// TIA Portal V17 export
// export: Created 2021-12-03T08:13:12.9041866Z, ExportSetting WithDefaults, DisplayName Totally Integrated Automation Portal, DisplayVersion V17, DisplayName TIA Portal Openness, DisplayVersion V17, DisplayName TIA Portal Version Control Interface, DisplayVersion V17, DisplayName STEP 7 Professional, DisplayVersion V17, DisplayName STEP 7 Safety, DisplayVersion V17, DisplayName WinCC Advanced, DisplayVersion V17
FUNCTION "FC_Safety_PerimeterCtrl" : Void   // FC300, F_FBD
VERSION : 0.1
// stored: AutoNumber false, IsIECCheckEnabled false, UDAEnableTagReadback false
BEGIN

REGION Network 1: Готовность к открытию
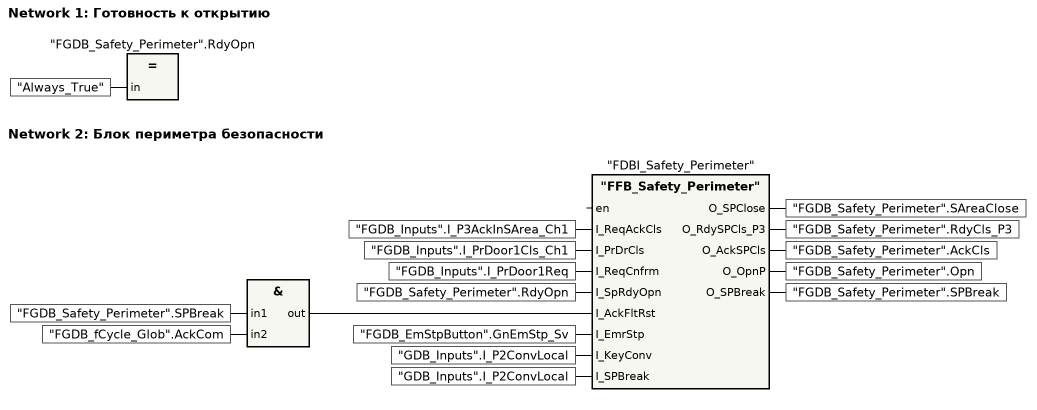
   "FGDB_Safety_Perimeter".RdyOpn := "Always_True";
END_REGION

REGION Network 2: Блок периметра безопасности
   "FDBI_Safety_Perimeter"(I_ReqAckCls := "FGDB_Inputs".I_P3AckInSArea_Ch1,   // "FFB_Safety_Perimeter"
                           I_PrDrCls := "FGDB_Inputs".I_PrDoor1Cls_Ch1,
                           I_ReqCnfrm := "FGDB_Inputs".I_PrDoor1Req,
                           I_SpRdyOpn := "FGDB_Safety_Perimeter".RdyOpn,
                           I_AckFltRst := "FGDB_Safety_Perimeter".SPBreak AND "FGDB_fCycle_Glob".AckCom,
                           I_EmrStp := "FGDB_EmStpButton".GnEmStp_Sv,
                           I_KeyConv := "GDB_Inputs".I_P2ConvLocal,
                           I_SPBreak := "GDB_Inputs".I_P2ConvLocal,
                           O_SPClose => "FGDB_Safety_Perimeter".SAreaClose,
                           O_RdySPCls_P3 => "FGDB_Safety_Perimeter".RdyCls_P3,
                           O_AckSPCls => "FGDB_Safety_Perimeter".AckCls,
                           O_OpnP => "FGDB_Safety_Perimeter".Opn,
                           O_SPBreak => "FGDB_Safety_Perimeter".SPBreak);
END_REGION
END_FUNCTION
